INTERFACE I_NodePrototypeEnumerator

END_INTERFACE

(* stored: Version 1.1.0.1, ProductVersion 3.1.4024.12
   Itf I_NodePrototypeEnumerator: Id {322daa39-a442-405f-98d3-0ec5cbf9d6c9} *)
